PROGRAM PRG_IM5K2_PPM
VAR
    {attribute 'pytmc' := '
        pv: IM5K2:PPM
        io: io
    '}
    {attribute 'TcLinkTo' := '.fbGige.iIlluminatorINT := TIIB[IM5K2-EL4004-E7]^AO Outputs Channel 1^Analog output;
                              .fbGige.bGigePower := TIIB[IM5K2-EL2004-E3]^Channel 2^Output;
                              .fbPowerMeter.iVoltageINT := TIIB[IM5K2-EL3062-E6]^AI Standard Channel 1^Value;
                              .fbPowerMeter.fbThermoCouple.bError := TIIB[IM5K2-EL3314-E4]^TC Inputs Channel 1^Status^Error;
                              .fbPowerMeter.fbThermoCouple.bUnderrange := TIIB[IM5K2-EL3314-E4]^TC Inputs Channel 1^Status^Underrange;
                              .fbPowerMeter.fbThermoCouple.bOverrange := TIIB[IM5K2-EL3314-E4]^TC Inputs Channel 1^Status^Overrange;
                              .fbPowerMeter.fbThermoCouple.iRaw := TIIB[IM5K2-EL3314-E4]^TC Inputs Channel 1^Value;
                              .fbYagThermoCouple.bError := TIIB[IM5K2-EL3314-E4]^TC Inputs Channel 2^Status^Error;
                              .fbYagThermoCouple.bUnderrange := TIIB[IM5K2-EL3314-E4]^TC Inputs Channel 2^Status^Underrange;
                              .fbYagThermoCouple.bOverrange := TIIB[IM5K2-EL3314-E4]^TC Inputs Channel 2^Status^Overrange;
                              .fbYagThermoCouple.iRaw := TIIB[IM5K2-EL3314-E4]^TC Inputs Channel 2^Value;
                              .fbFlowMeter.iRaw := TIIB[IM5K2-EL3052-E5]^AI Standard Channel 1^Value'}
    fbIM5K2: FB_PPM;
END_VAR


fbIM5K2.stOut.fPosition := -8.92;
fbIM5K2.stOut.bUseRawCounts := FALSE;
fbIM5K2.stOut.bValid := TRUE;
fbIM5K2.stOut.stPMPS.sPmpsState := 'IM5K2:PPM-OUT';

fbIM5K2.stPower.fPosition := -48.02;
fbIM5K2.stPower.bUseRawCounts := FALSE;
fbIM5K2.stPower.bValid := TRUE;
fbIM5K2.stPower.stPMPS.sPmpsState := 'IM5K2:PPM-POWERMETER';

fbIM5K2.stYag1.fPosition := -72.02;
fbIM5K2.stYag1.bUseRawCounts := FALSE;
fbIM5K2.stYag1.bValid := TRUE;
fbIM5K2.stYag1.stPMPS.sPmpsState := 'IM5K2:PPM-YAG1';

fbIM5K2.stYag2.fPosition := -98.03;
fbIM5K2.stYag2.bUseRawCounts := FALSE;
fbIM5K2.stYag2.bValid := TRUE;
fbIM5K2.stYag2.stPMPS.sPmpsState := 'IM5K2:PPM-YAG2';

fbIM5K2(
    fbArbiter := GVL.fbArbiter2,
    fbFFHWO := GVL.fbFastFaultOutput2,
    stYStage := Main.M14,
    sDeviceName := 'IM5K2:PPM',
    sTransitionKey := 'IM5K2:PPM-TRANSITION',
    bEnableMotion := TRUE,
    bEnableBeamParams := TRUE,
    bEnablePositionLimits := TRUE,
    fFlowOffset := 0.0,
);

END_PROGRAM

(* stored: Version 1.1.0.1, ProductVersion 3.1.4022.18
   POU PRG_IM5K2_PPM: Id {ce83f37e-c4d6-4a90-b3a1-93181924ae90}, SpecialFunc None *)
